PROGRAM P_Demo_F_BA_TimeMerge
VAR
    argStTime1                     : ST_BA_Time                    ; // stTime1
    argStTime2                     : ST_BA_Time                    ; // stTime2
    fnReturn                       : ST_BA_Time; // 返回值
END_VAR

// =============================================================================
// Tc3_BA2_Common.F_BA_TimeMerge 演示程序
// =============================================================================
// 场景：从用户输入的 4 个数字字段构造时间。
//
// 价值：一行替代字段赋值。
//
// 验证：登录 PLC 后，按例程内变量在线写值；监视输出 / 返回值，结合 §1 功能
//       简述的预期行为对照（详见配套 .md 文档 §7 业务场景）。
//
// 验证步骤：
//   1. 右键 PLC 项目下 POUs 文件夹 → Add → Existing Item → 选本 .TcPOU 文件
//   2. 引用 Tc3_BA2_Common（References → Add library）
//   3. 编译 → 登录 → 运行；按上方『验证』指引在线写值观察
// =============================================================================

fnReturn := F_BA_TimeMerge(
    stTime1                  := argStTime1,
    stTime2                  := argStTime2
);

END_PROGRAM

(* stored: Version 1.1.0.1, ProductVersion 3.1.4024.5
   POU P_Demo_F_BA_TimeMerge: Id {ab19f313-9ede-50a9-a3db-42eb545feecf}, SpecialFunc None *)
